{attribute 'GeneratedUsingTerminal: EL1512-0000-0017'}
{attribute addProperty BoxType "EL1512-0000-0017"}
{attribute addProperty Id "StatusAT %I*Status_8AD1B54B4Counter_valueAT %I*UDINT4"}
{attribute addProperty CRC "1426009886"}
{attribute addProperty Size "8"}
TYPE CNT_Inputs_Channel_54FF2F1E EXTENDS InputBase_8311D824 :
STRUCT
	{attribute addProperty Name "Status"}
	Status AT %I* : Status_8AD1B54B;
	{attribute addProperty Name "Counter_value"}
	Counter_value AT %I* : UDINT;
END_STRUCT
END_TYPE

(* stored: Version 1.2.0.0, ProductVersion 3.1.4024.9
   DUT CNT_Inputs_Channel_54FF2F1E: Id {995a6c9a-cc1d-492e-9be0-9aa12b210152} *)
